// TwinCAT 3 PLC project Test
// ProgramVersion: 3.1.4023.0
// libraries:
//   Tc2_Standard, * (Beckhoff Automation GmbH)
//   Tc2_System, * (Beckhoff Automation GmbH)
//   Tc3_Module, * (Beckhoff Automation GmbH)
// project tree:
//   / PlcTask.TcTTO
//   POUs/ MAIN.TcPOU
// real-time tasks:
//   TASK PlcTask: cycle T#10ms, priority 20, ADS port 350

CONFIGURATION Test
    RESOURCE PLC ON TwinCAT3
        TASK PlcTask(INTERVAL := T#10ms, PRIORITY := 20);
        PROGRAM MAIN WITH PlcTask : MAIN;
    END_RESOURCE
END_CONFIGURATION

// ---- POUs/MAIN.TcPOU
PROGRAM MAIN
VAR
	sintVal 	AT 	%MB0 	: SINT;
	intVal		AT	%MB8 	: INT;
	dintVal 	AT	%MB16 	: DINT;
	boolVal		AT	%MX24.0	: BOOL;
	floatVal 	AT	%MB32	: REAL;
	doubleVal	AT	%MB40	: LREAL;
	stringVal	AT	%MB48	: STRING;
END_VAR

END_PROGRAM
